TYPE
LRK_typeCamStatus :
STRUCT
    cam                      : INT;
    control                  : BOOL;
    error                    : BOOL;
    restartActive            : BOOL;
    onlineStartValuesChanged : BOOL;
    camDataChanged           : BOOL;
    interpolated             : BOOL;
    inInterpolation          : BOOL;
    restartDone              : BOOL;
    restartBusy              : BOOL;
    restartCommandAborted    : BOOL;
    restartError             : BOOL;
    restartErrorId           : WORD;
    interpolateCamDone       : BOOL;
    interpolateCamBusy       : BOOL;
    interpolateCamError      : BOOL;
    interpolateCamErrorId    : WORD;
    startLeadingValue        : LREAL;
    endLeadingValue          : LREAL;
END_STRUCT
END_TYPE

(* stored: Version 1.1.0.1
   DUT LRK_typeCamStatus: Id {9308c777-6fc3-4237-bbf6-45576c4db79a} *)
